Fanuc KAREL source: ka00079.KL

-- PROVISIONAL review KL for V1013-1; original PC SHA256 d8bdf71f5657215fe684086402645263a82e1bd368636e8ebd79ca9890bf67e9
-- Incomplete behavior may be omitted. Consult companion uncertainty JSON. Do not deploy.
PROGRAM KA00079
%NOLOCKGROUP
-- UNRESOLVED_DECL SRC type=000106
-- UNRESOLVED_DECL DST type=000106
BEGIN
  -- UNRESOLVED_PC offsets 5-20; opcodes 2E,22,32,35
  -- UNRESOLVED_PC offsets 25-40; opcodes 49,4A
  -- UNRESOLVED_PC offsets 45-49; opcodes 7F
END KA00079
